Omron CX-Programmer project NewProject (CX-Programmer 9.73)

# PLC NewPLC1: CJ2M CPU11
I/O table (CPU CJ2M-CPU11): rack 0 slot 0 CJ1W-ID211; rack 0 slot 1 CJ1W-OC211; rack 0 slot 2 CJ1W-ETN21(ETN21Mode)

## Global symbols (name address type ; comment)
T0000 BOOL  ; timer
T0010 BOOL  ; Emergencia Cilindro recuo
T0011 BOOL  ; Emergencia ciclindro avanço
T0015 BOOL  ; Emergencia Vacuo pneumatico movimento para cima
T0016 BOOL  ; Emergencia Vacuo pneumatico movimento para baixo
T0017 BOOL  ; Emergencia Vacuo pneumatico movimento para tras
T0018 BOOL  ; Emergencia Vacuo pneumatico movimento para frente
W1.00 BOOL  ; COm1
W1.01 BOOL  ; Com2
Outra_vez 202.03 BOOL

## Program NewProgram1 (cyclic task 0)
Local symbols
A1_APnV 1.07 BOOL  ; Avanço Pneumatico Vácuo
A1_BPnV 1.15 BOOL  ; Baixa Pneumatico Vácuo
A1_Chave 0.02 BOOL
A1_MT 1.06 BOOL  ; Motor Tapete
A1_PI 1.14 BOOL  ; Pneumatico Inicio
A1_RPnV 1.10 BOOL  ; Recua Pneumatico Vácuo
A1_Reset 0.03 BOOL
A1_SP 1.11 BOOL  ; Stop Peça
A1_S_C 0.13 BOOL  ; Sensor Leitura Cor
A1_S_C_A2 D100.05 BOOL  ; Transmisao Sensor Leitura Cor A1 para A2
A1_S_FT 0.14 BOOL  ; Sensor Fim Tapete
A1_S_FT_A2 D100.06 BOOL  ; Transmisao Sensor Fim Tapete A1 para A2
A1_S_IT 0.08 BOOL  ; Sensor Inicio Tapete
A1_S_IT_A2 D100.04 BOOL  ; Transmisao Sensor inicio Tapete A1 para A2
A1_S_PB 0.06 BOOL  ; Sensor Deteta Peça Base
A1_S_PnF 0.04 BOOL  ; Sensor Pneumático Frente
A1_S_PnT 0.05 BOOL  ; Sensor Pneumático Tras
A1_S_V 0.12 BOOL  ; Sensor Vácuo
A1_S_VPnC 0.11 BOOL  ; Sensor Vácuo Pneumatico cima
A1_S_VPnF 0.09 BOOL  ; Sensor Vácuo Pneumatico Frente
A1_S_VPnT 0.10 BOOL  ; Sensor Vácuo Pneumatico Tras
A1_Start 0.00 BOOL
A1_Stop 0.01 BOOL
A1_V 1.12 BOOL  ; Vácuo
A2_A1_MT D1.02 BOOL  ; Comunicaçao A2 para A1 para ativar motor tapete
A2_S_PR D1.01 BOOL  ; Sensor Posição Recolha (automato 2)
Again 202.02 BOOL
Cilindro_Base D1.03 BOOL  ; Manual
Cilindro_Tampa_Back D1.05 BOOL  ; Manual
Cilindro_Tampa_Down D1.06 BOOL  ; Manual
Cilindro_Tampa_Front D1.04 BOOL  ; Manual
Control_Array 205 UINT
Count 206 UINT
E_10 200.05 BOOL
E_11 200.06 BOOL
E_12 200.07 BOOL
E_13 200.08 BOOL
E_20 200.09 BOOL
E_21 200.10 BOOL
E_22 200.11 BOOL
E_23 200.12 BOOL
E_24 200.03 BOOL
E_25 200.13 BOOL
E_26 200.14 BOOL
E_27 200.15 BOOL
E_28 201.00 BOOL
E_30 201.03 BOOL
E_31 201.04 BOOL
E_32 201.05 BOOL
E_33 201.06 BOOL  ; Modulo Vacuo
E_34 201.07 BOOL
E_35 201.08 BOOL
E_36 201.09 BOOL
E_37 201.10 BOOL  ; Modulo Vacuo
E_38 201.11 BOOL
E_39 201.12 BOOL
E_40 201.13 BOOL  ; Modulo Vacuo
E_41 201.14 BOOL
E_42 200.02 BOOL
E_45 201.01 BOOL
E_46 201.02 BOOL
Emergencia_Cilindro_recuo D102.00 BOOL
Emergencia_Vacuo_pneumatico_movimento_para_baixo D102.03 BOOL
Emergencia_Vacuo_pneumatico_movimento_para_cima D102.02 BOOL
Emergencia_Vacuo_pneumatico_movimento_para_frente D102.05 BOOL
Emergencia_Vacuo_pneumatico_movimento_para_tras D102.04 BOOL
Emergencia_ciclindro_avanço D102.01 BOOL
Emergencia_peca_vacuo_nao_detetada D102.06 BOOL
Execute D1.00 BOOL
MT_Force_Down 202.03 BOOL
Reset D100.02 BOOL
Start D100.00 BOOL
Stop D100.01 BOOL
Tapete D1.09 BOOL  ; Manual
Travão_Montagem D1.08 BOOL  ; Manual
Vácuo D1.07 BOOL  ; Manual

### Section Inicialization

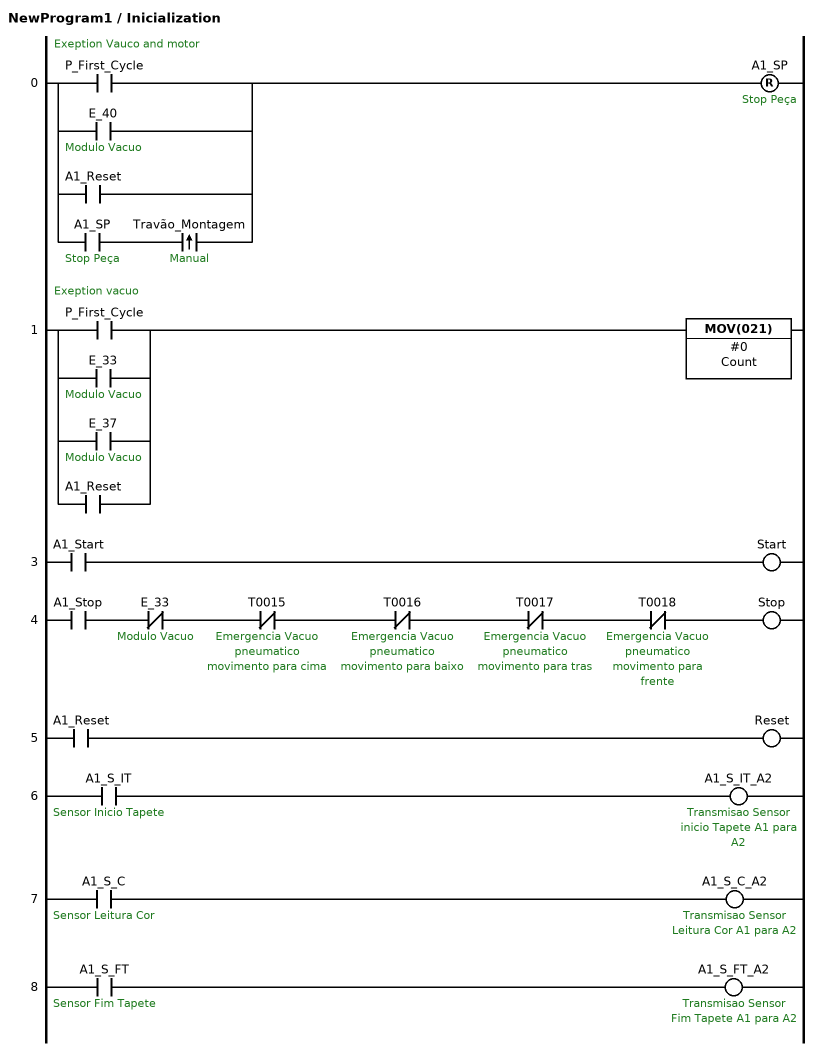
; rung 0: Exeption Vauco and motor
LD P_First_Cycle
OR E_40  ; Modulo Vacuo
OR A1_Reset
LD A1_SP  ; Stop Peça
@AND Travão_Montagem  ; Manual
ORLD
RSET A1_SP  ; Stop Peça
; rung 1: Exeption vacuo
LD P_First_Cycle
OR E_33  ; Modulo Vacuo
OR E_37  ; Modulo Vacuo
OR A1_Reset
MOV(021) #0 Count
; rung 3
LD A1_Start
OUT Start
; rung 4
LD A1_Stop
ANDNOT E_33  ; Modulo Vacuo
ANDNOT T0015  ; Emergencia Vacuo pneumatico movimento para cima
ANDNOT T0016  ; Emergencia Vacuo pneumatico movimento para baixo
ANDNOT T0017  ; Emergencia Vacuo pneumatico movimento para tras
ANDNOT T0018  ; Emergencia Vacuo pneumatico movimento para frente
OUT Stop
; rung 5
LD A1_Reset
OUT Reset
; rung 6
LD A1_S_IT  ; Sensor Inicio Tapete
OUT A1_S_IT_A2  ; Transmisao Sensor inicio Tapete A1 para A2
; rung 7
LD A1_S_C  ; Sensor Leitura Cor
OUT A1_S_C_A2  ; Transmisao Sensor Leitura Cor A1 para A2
; rung 8
LD A1_S_FT  ; Sensor Fim Tapete
OUT A1_S_FT_A2  ; Transmisao Sensor Fim Tapete A1 para A2

### Section Init

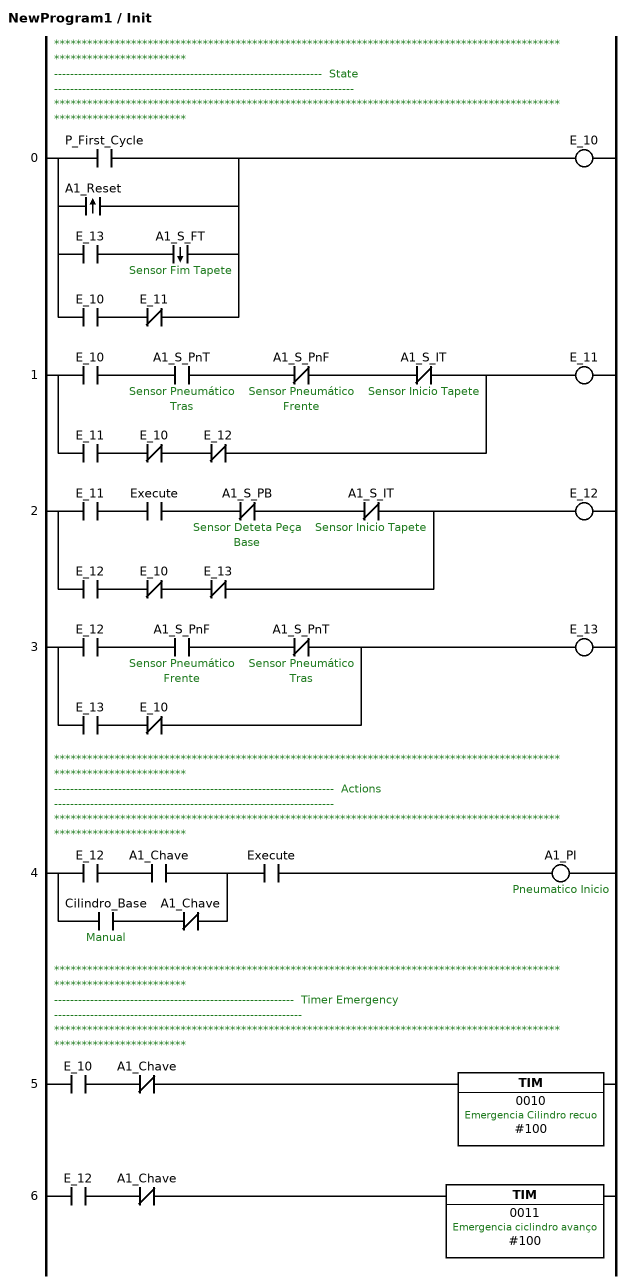
; rung 0: ******************************************************************************************************************** / -------------------------------------------------------------------  State  --------------------------------------------------------------------------- / ********************************************************************************************************************
LD P_First_Cycle
@OR A1_Reset
LD E_13
%AND A1_S_FT  ; Sensor Fim Tapete
ORLD
LD E_10
ANDNOT E_11
ORLD
OUT E_10
; rung 1
LD E_10
AND A1_S_PnT  ; Sensor Pneumático Tras
ANDNOT A1_S_PnF  ; Sensor Pneumático Frente
ANDNOT A1_S_IT  ; Sensor Inicio Tapete
LD E_11
ANDNOT E_10
ANDNOT E_12
ORLD
OUT E_11
; rung 2
LD E_11
AND Execute
ANDNOT A1_S_PB  ; Sensor Deteta Peça Base
ANDNOT A1_S_IT  ; Sensor Inicio Tapete
LD E_12
ANDNOT E_10
ANDNOT E_13
ORLD
OUT E_12
; rung 3
LD E_12
AND A1_S_PnF  ; Sensor Pneumático Frente
ANDNOT A1_S_PnT  ; Sensor Pneumático Tras
LD E_13
ANDNOT E_10
ORLD
OUT E_13
; rung 4: ******************************************************************************************************************** / ----------------------------------------------------------------------  Actions ---------------------------------------------------------------------- / ********************************************************************************************************************
LD E_12
AND A1_Chave
LD Cilindro_Base  ; Manual
ANDNOT A1_Chave
ORLD
AND Execute
OUT A1_PI  ; Pneumatico Inicio
; rung 5: ******************************************************************************************************************** / ------------------------------------------------------------  Timer Emergency  -------------------------------------------------------------- / ********************************************************************************************************************
LD E_10
ANDNOT A1_Chave
TIM 0010 #100  ; Emergencia Cilindro recuo
; rung 6
LD E_12
ANDNOT A1_Chave
TIM 0011 #100  ; Emergencia ciclindro avanço

### Section Belt

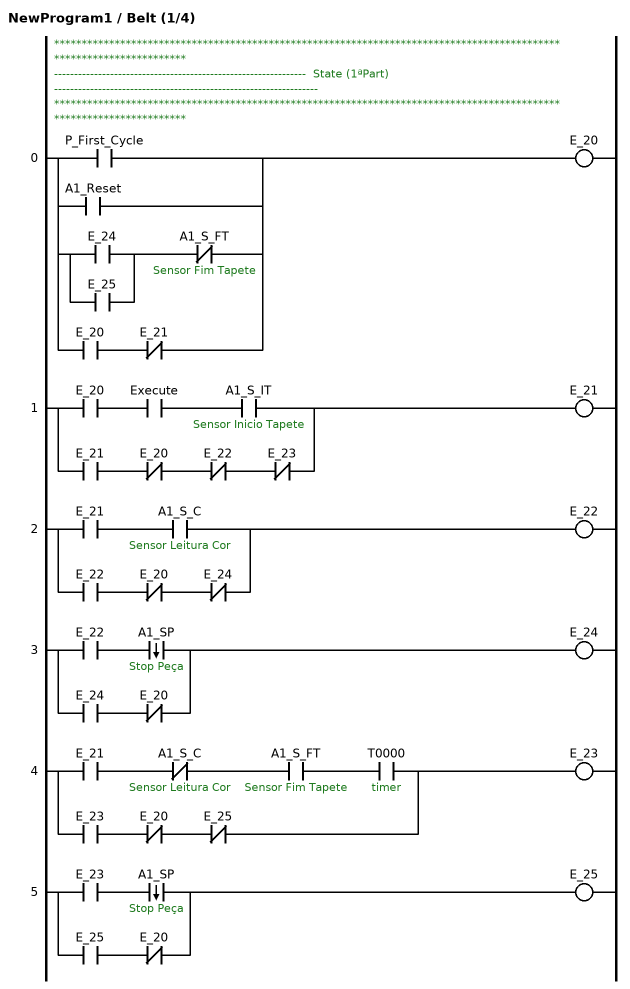
; rung 0: ******************************************************************************************************************** / ---------------------------------------------------------------  State (1ªPart)  ------------------------------------------------------------------ / ********************************************************************************************************************
LD P_First_Cycle
OR A1_Reset
LD E_24
OR E_25
ANDNOT A1_S_FT  ; Sensor Fim Tapete
ORLD
LD E_20
ANDNOT E_21
ORLD
OUT E_20
; rung 1
LD E_20
AND Execute
AND A1_S_IT  ; Sensor Inicio Tapete
LD E_21
ANDNOT E_20
ANDNOT E_22
ANDNOT E_23
ORLD
OUT E_21
; rung 2
LD E_21
AND A1_S_C  ; Sensor Leitura Cor
LD E_22
ANDNOT E_20
ANDNOT E_24
ORLD
OUT E_22
; rung 3
LD E_22
%AND A1_SP  ; Stop Peça
LD E_24
ANDNOT E_20
ORLD
OUT E_24
; rung 4
LD E_21
ANDNOT A1_S_C  ; Sensor Leitura Cor
AND A1_S_FT  ; Sensor Fim Tapete
AND T0000  ; timer
LD E_23
ANDNOT E_20
ANDNOT E_25
ORLD
OUT E_23
; rung 5
LD E_23
%AND A1_SP  ; Stop Peça
LD E_25
ANDNOT E_20
ORLD
OUT E_25

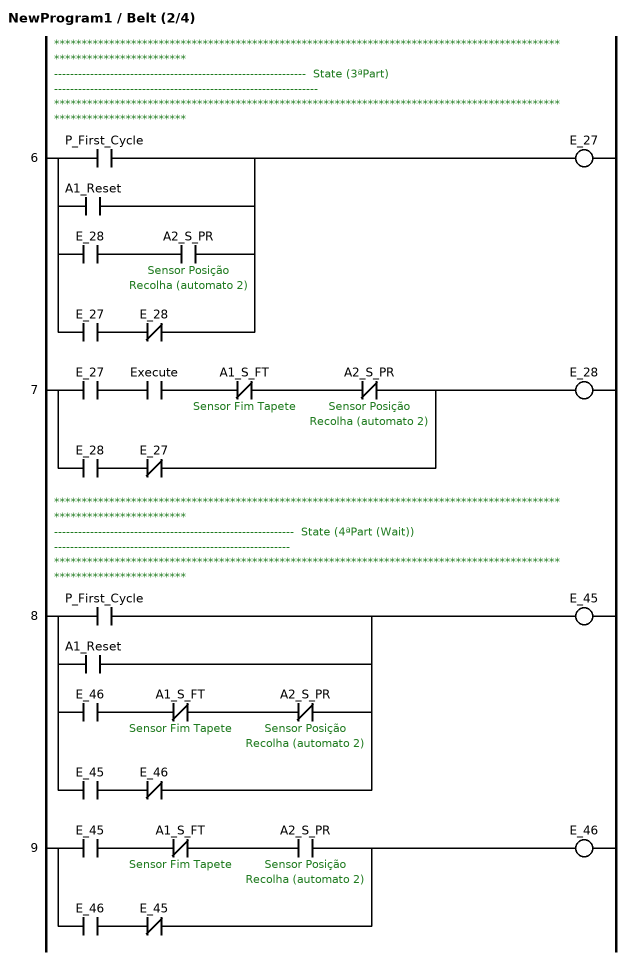
; rung 6: ******************************************************************************************************************** / ---------------------------------------------------------------  State (3ªPart)  ------------------------------------------------------------------ / ********************************************************************************************************************
LD P_First_Cycle
OR A1_Reset
LD E_28
AND A2_S_PR  ; Sensor Posição Recolha (automato 2)
ORLD
LD E_27
ANDNOT E_28
ORLD
OUT E_27
; rung 7
LD E_27
AND Execute
ANDNOT A1_S_FT  ; Sensor Fim Tapete
ANDNOT A2_S_PR  ; Sensor Posição Recolha (automato 2)
LD E_28
ANDNOT E_27
ORLD
OUT E_28
; rung 8: ******************************************************************************************************************** / ------------------------------------------------------------  State (4ªPart (Wait))  ----------------------------------------------------------- / ********************************************************************************************************************
LD P_First_Cycle
OR A1_Reset
LD E_46
ANDNOT A1_S_FT  ; Sensor Fim Tapete
ANDNOT A2_S_PR  ; Sensor Posição Recolha (automato 2)
ORLD
LD E_45
ANDNOT E_46
ORLD
OUT E_45
; rung 9
LD E_45
ANDNOT A1_S_FT  ; Sensor Fim Tapete
AND A2_S_PR  ; Sensor Posição Recolha (automato 2)
LD E_46
ANDNOT E_45
ORLD
OUT E_46

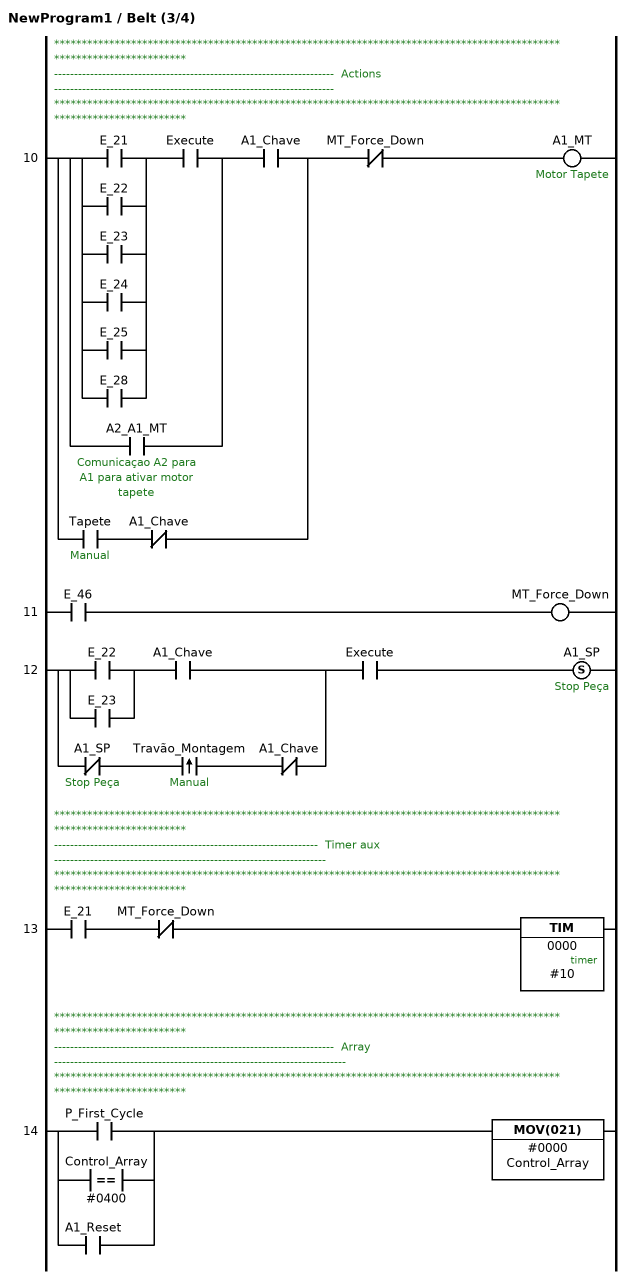
; rung 10: ******************************************************************************************************************** / ----------------------------------------------------------------------  Actions ---------------------------------------------------------------------- / ********************************************************************************************************************
LD E_21
OR E_22
OR E_23
OR E_24
OR E_25
OR E_28
AND Execute
OR A2_A1_MT  ; Comunicaçao A2 para A1 para ativar motor tapete
AND A1_Chave
LD Tapete  ; Manual
ANDNOT A1_Chave
ORLD
ANDNOT MT_Force_Down
OUT A1_MT  ; Motor Tapete
; rung 11
LD E_46
OUT MT_Force_Down
; rung 12
LD E_22
OR E_23
AND A1_Chave
LDNOT A1_SP  ; Stop Peça
@AND Travão_Montagem  ; Manual
ANDNOT A1_Chave
ORLD
AND Execute
SET A1_SP  ; Stop Peça
; rung 13: ******************************************************************************************************************** / ------------------------------------------------------------------  Timer aux  -------------------------------------------------------------------- / ********************************************************************************************************************
LD E_21
ANDNOT MT_Force_Down
TIM 0000 #10  ; timer
; rung 14: ******************************************************************************************************************** / ----------------------------------------------------------------------  Array  ------------------------------------------------------------------------- / ********************************************************************************************************************
LD P_First_Cycle
OR=(300) Control_Array #0400
OR A1_Reset
MOV(021) #0000 Control_Array

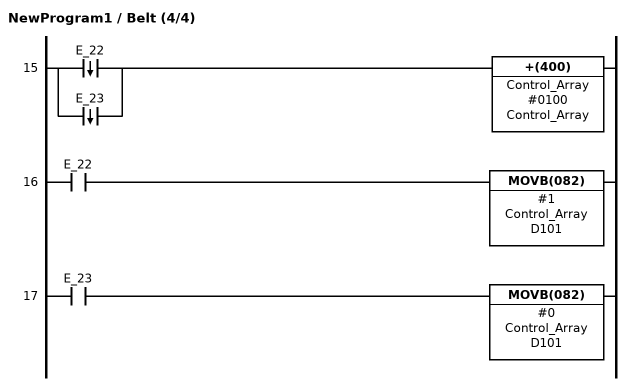
; rung 15
%LD E_22
%OR E_23
+(400) Control_Array #0100 Control_Array
; rung 16
LD E_22
MOVB(082) #1 Control_Array D101
; rung 17
LD E_23
MOVB(082) #0 Control_Array D101

### Section Vacuum

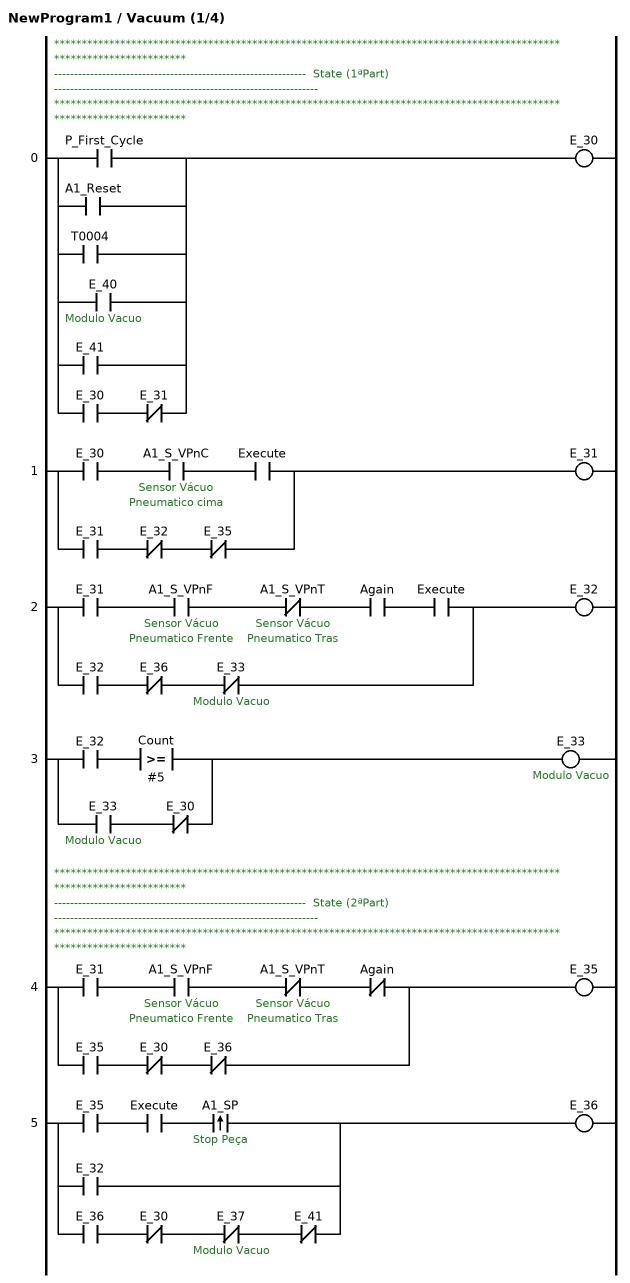
; rung 0: ******************************************************************************************************************** / ---------------------------------------------------------------  State (1ªPart)  ------------------------------------------------------------------ / ********************************************************************************************************************
LD P_First_Cycle
OR A1_Reset
OR T0004
OR E_40  ; Modulo Vacuo
OR E_41
LD E_30
ANDNOT E_31
ORLD
OUT E_30
; rung 1
LD E_30
AND A1_S_VPnC  ; Sensor Vácuo Pneumatico cima
AND Execute
LD E_31
ANDNOT E_32
ANDNOT E_35
ORLD
OUT E_31
; rung 2
LD E_31
AND A1_S_VPnF  ; Sensor Vácuo Pneumatico Frente
ANDNOT A1_S_VPnT  ; Sensor Vácuo Pneumatico Tras
AND Again
AND Execute
LD E_32
ANDNOT E_36
ANDNOT E_33  ; Modulo Vacuo
ORLD
OUT E_32
; rung 3
LD E_32
AND>=(325) Count #5
LD E_33  ; Modulo Vacuo
ANDNOT E_30
ORLD
OUT E_33  ; Modulo Vacuo
; rung 4: ******************************************************************************************************************** / ---------------------------------------------------------------  State (2ªPart)  ------------------------------------------------------------------ / ********************************************************************************************************************
LD E_31
AND A1_S_VPnF  ; Sensor Vácuo Pneumatico Frente
ANDNOT A1_S_VPnT  ; Sensor Vácuo Pneumatico Tras
ANDNOT Again
LD E_35
ANDNOT E_30
ANDNOT E_36
ORLD
OUT E_35
; rung 5
LD E_35
AND Execute
@AND A1_SP  ; Stop Peça
OR E_32
LD E_36
ANDNOT E_30
ANDNOT E_37  ; Modulo Vacuo
ANDNOT E_41
ORLD
OUT E_36

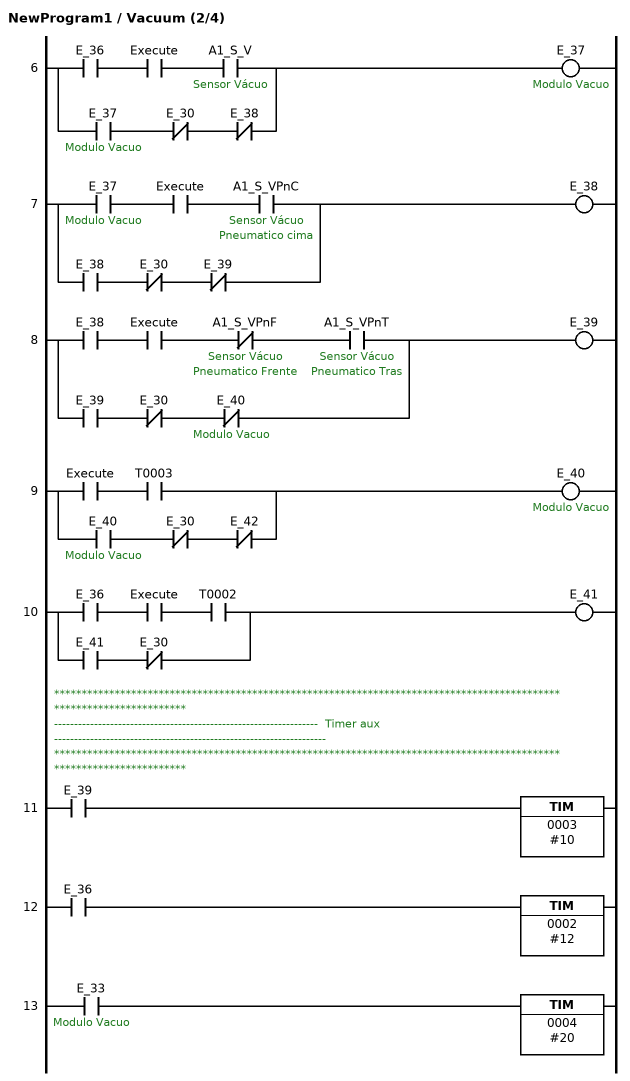
; rung 6
LD E_36
AND Execute
AND A1_S_V  ; Sensor Vácuo
LD E_37  ; Modulo Vacuo
ANDNOT E_30
ANDNOT E_38
ORLD
OUT E_37  ; Modulo Vacuo
; rung 7
LD E_37  ; Modulo Vacuo
AND Execute
AND A1_S_VPnC  ; Sensor Vácuo Pneumatico cima
LD E_38
ANDNOT E_30
ANDNOT E_39
ORLD
OUT E_38
; rung 8
LD E_38
AND Execute
ANDNOT A1_S_VPnF  ; Sensor Vácuo Pneumatico Frente
AND A1_S_VPnT  ; Sensor Vácuo Pneumatico Tras
LD E_39
ANDNOT E_30
ANDNOT E_40  ; Modulo Vacuo
ORLD
OUT E_39
; rung 9
LD Execute
AND T0003
LD E_40  ; Modulo Vacuo
ANDNOT E_30
ANDNOT E_42
ORLD
OUT E_40  ; Modulo Vacuo
; rung 10
LD E_36
AND Execute
AND T0002
LD E_41
ANDNOT E_30
ORLD
OUT E_41
; rung 11: ******************************************************************************************************************** / ------------------------------------------------------------------  Timer aux  -------------------------------------------------------------------- / ********************************************************************************************************************
LD E_39
TIM 0003 #10
; rung 12
LD E_36
TIM 0002 #12
; rung 13
LD E_33  ; Modulo Vacuo
TIM 0004 #20

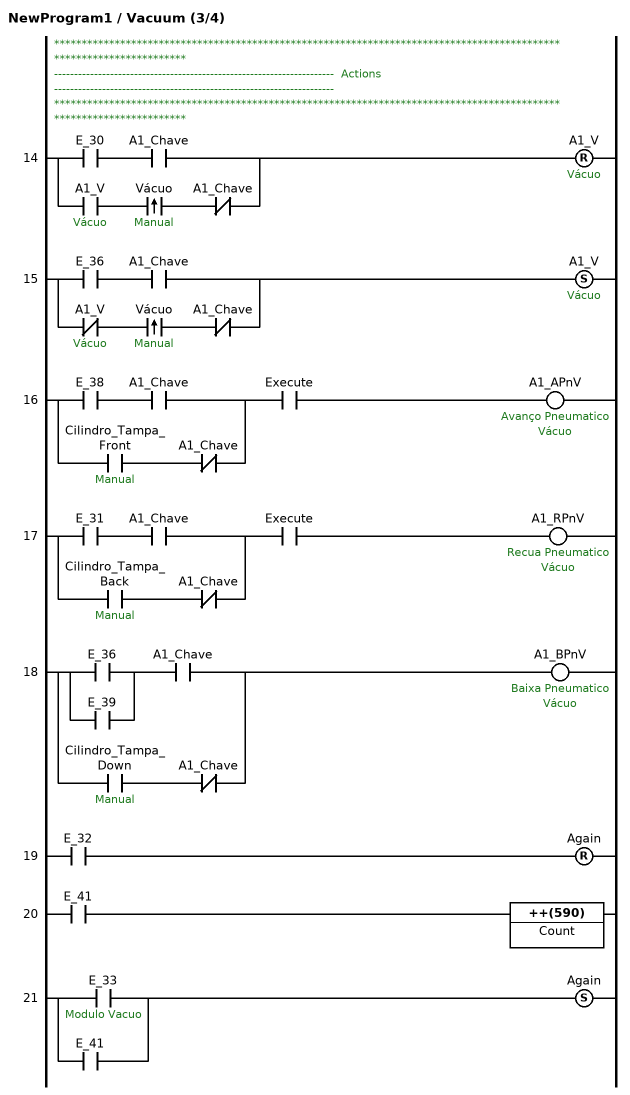
; rung 14: ******************************************************************************************************************** / ----------------------------------------------------------------------  Actions ---------------------------------------------------------------------- / ********************************************************************************************************************
LD E_30
AND A1_Chave
LD A1_V  ; Vácuo
@AND Vácuo  ; Manual
ANDNOT A1_Chave
ORLD
RSET A1_V  ; Vácuo
; rung 15
LD E_36
AND A1_Chave
LDNOT A1_V  ; Vácuo
@AND Vácuo  ; Manual
ANDNOT A1_Chave
ORLD
SET A1_V  ; Vácuo
; rung 16
LD E_38
AND A1_Chave
LD Cilindro_Tampa_Front  ; Manual
ANDNOT A1_Chave
ORLD
AND Execute
OUT A1_APnV  ; Avanço Pneumatico Vácuo
; rung 17
LD E_31
AND A1_Chave
LD Cilindro_Tampa_Back  ; Manual
ANDNOT A1_Chave
ORLD
AND Execute
OUT A1_RPnV  ; Recua Pneumatico Vácuo
; rung 18
LD E_36
OR E_39
AND A1_Chave
LD Cilindro_Tampa_Down  ; Manual
ANDNOT A1_Chave
ORLD
OUT A1_BPnV  ; Baixa Pneumatico Vácuo
; rung 19
LD E_32
RSET Again
; rung 20
LD E_41
++(590) Count
; rung 21
LD E_33  ; Modulo Vacuo
OR E_41
SET Again

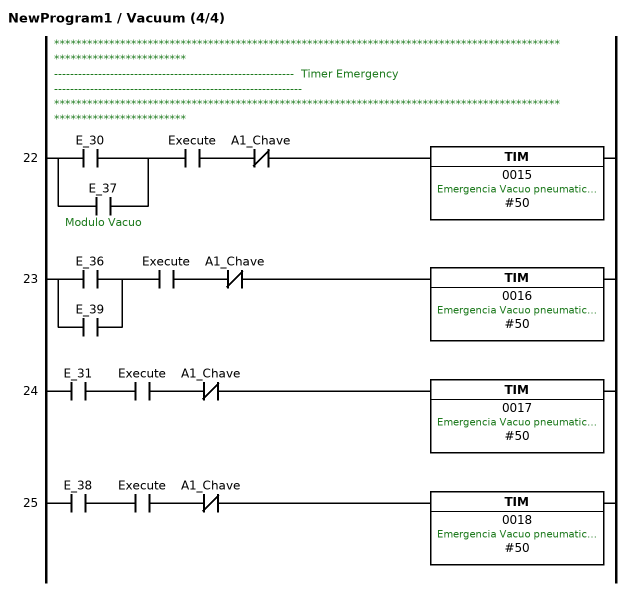
; rung 22: ******************************************************************************************************************** / ------------------------------------------------------------  Timer Emergency  -------------------------------------------------------------- / ********************************************************************************************************************
LD E_30
OR E_37  ; Modulo Vacuo
AND Execute
ANDNOT A1_Chave
TIM 0015 #50  ; Emergencia Vacuo pneumatico movimento para cima
; rung 23
LD E_36
OR E_39
AND Execute
ANDNOT A1_Chave
TIM 0016 #50  ; Emergencia Vacuo pneumatico movimento para baixo
; rung 24
LD E_31
AND Execute
ANDNOT A1_Chave
TIM 0017 #50  ; Emergencia Vacuo pneumatico movimento para tras
; rung 25
LD E_38
AND Execute
ANDNOT A1_Chave
TIM 0018 #50  ; Emergencia Vacuo pneumatico movimento para frente

### Section Emergency

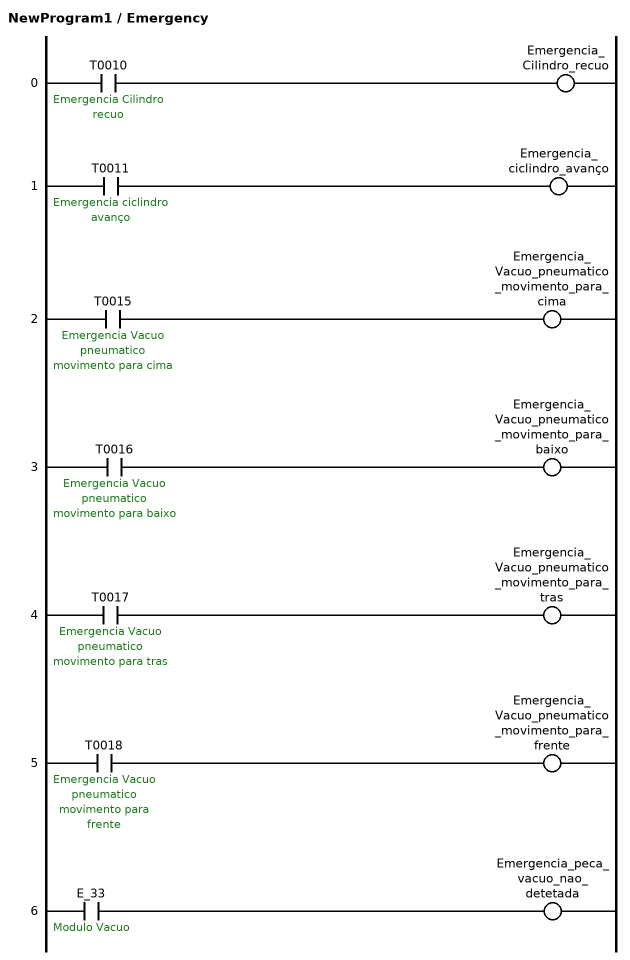
; rung 0
LD T0010  ; Emergencia Cilindro recuo
OUT Emergencia_Cilindro_recuo
; rung 1
LD T0011  ; Emergencia ciclindro avanço
OUT Emergencia_ciclindro_avanço
; rung 2
LD T0015  ; Emergencia Vacuo pneumatico movimento para cima
OUT Emergencia_Vacuo_pneumatico_movimento_para_cima
; rung 3
LD T0016  ; Emergencia Vacuo pneumatico movimento para baixo
OUT Emergencia_Vacuo_pneumatico_movimento_para_baixo
; rung 4
LD T0017  ; Emergencia Vacuo pneumatico movimento para tras
OUT Emergencia_Vacuo_pneumatico_movimento_para_tras
; rung 5
LD T0018  ; Emergencia Vacuo pneumatico movimento para frente
OUT Emergencia_Vacuo_pneumatico_movimento_para_frente
; rung 6
LD E_33  ; Modulo Vacuo
OUT Emergencia_peca_vacuo_nao_detetada

### Section END
; rung 0
END(001)